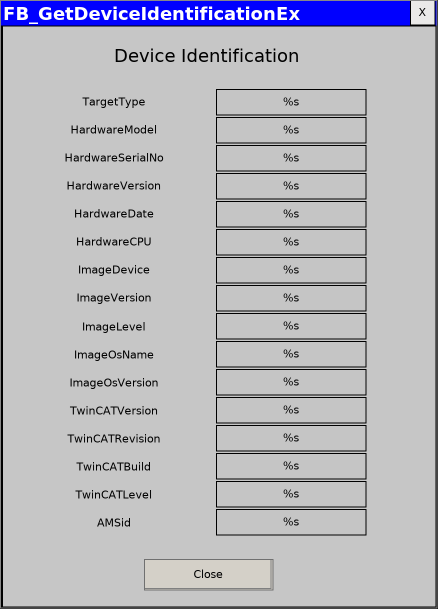
VISUALIZATION dialogDeviceInfo  // 438x609
    Rectangle (0,0 438x609)
        OnMouseClick: CloseDialog Dialog=dialogDeviceInfo, Result=OK, NumpadKeypadSet=True
    Button (144,559 129x31), "Close"
        OnMouseClick: CloseDialog Dialog=dialogDeviceInfo, Result=None, NumpadKeypadSet=True
    Rectangle (0,0 438x26), "FB_GetDeviceIdentificationEx"
    Rectangle (410,0 25x25), "X"
        OnMouseClick: CloseDialog Dialog=dialogDeviceInfo, Result=Cancel, NumpadKeypadSet=True
    Rectangle (216,89 150x26), "%s", text variable: System.sysDeviceInfo.strTargetType
    Label (16,89 196x26), "TargetType"
    Label (16,117 196x26), "HardwareModel"
    Rectangle (216,117 150x26), "%s", text variable: System.sysDeviceInfo.strHardwareModel
    Rectangle (216,145 150x26), "%s", text variable: System.sysDeviceInfo.strHardwareSerialNo
    Label (16,145 196x26), "HardwareSerialNo"
    Label (16,173 196x26), "HardwareVersion"
    Rectangle (216,173 150x26), "%s", text variable: System.sysDeviceInfo.strHardwareVersion
    Rectangle (216,201 150x26), "%s", text variable: System.sysDeviceInfo.strHardwareDate
    Label (16,201 196x26), "HardwareDate"
    Label (16,229 196x26), "HardwareCPU"
    Rectangle (216,229 150x26), "%s", text variable: System.sysDeviceInfo.strHardwareCPU
    Rectangle (216,257 150x26), "%s", text variable: System.sysDeviceInfo.strImageDevice
    Label (16,257 196x26), "ImageDevice"
    Label (16,285 196x26), "ImageVersion"
    Rectangle (216,285 150x26), "%s", text variable: System.sysDeviceInfo.strImageVersion
    Rectangle (216,313 150x26), "%s", text variable: System.sysDeviceInfo.strImageLevel
    Label (16,314 196x26), "ImageLevel"
    Label (16,342 196x26), "ImageOsName"
    Rectangle (216,341 150x26), "%s", text variable: System.sysDeviceInfo.strImageOsName
    Rectangle (216,369 150x26), "%s", text variable: System.sysDeviceInfo.strImageOsVersion
    Label (16,370 196x26), "ImageOsVersion"
    Label (16,398 196x26), "TwinCATVersion"
    Rectangle (216,397 150x26), "%s", text variable: System.sysDeviceInfo.strTwinCATVersion
    Rectangle (216,425 150x26), "%s", text variable: System.sysDeviceInfo.strTwinCATRevision
    Label (16,426 196x26), "TwinCATRevision"
    Rectangle (216,453 150x26), "%s", text variable: System.sysDeviceInfo.strTwinCATBuild
    Label (16,454 196x26), "TwinCATBuild"
    Label (16,482 196x26), "TwinCATLevel"
    Rectangle (216,481 150x26), "%s", text variable: System.sysDeviceInfo.strTwinCATLevel
    Label (16,510 196x26), "AMSid"
    Rectangle (216,509 150x26), "%s", text variable: System.sysDeviceInfo.strAmsNetId
    Label (109,43 196x26), "Device Identification"
END_VISUALIZATION

(* stored: Version 1.1.0.1, ProductVersion 3.1.4024.12
   Visu dialogDeviceInfo: Id {fd487386-f792-420e-9f9e-c8a7082e9218} *)
